{attribute 'GeneratedUsingTerminal: EK1100-0000-0018'}
{attribute addProperty BoxType "EK1100-0000-0018"}
{attribute addProperty Id "Beckhoff_APS1xxxEK1122Beckhoff_APS1xxxEK1122_47B4CB21266A_0002_APS1003_5000_0016APS1003_748FE0C1320"}
{attribute addProperty CRC "3524367647"}
{attribute addProperty Size "586"}
TYPE Beckhoff_APS1xxx_D211951F EXTENDS EK1100_AB5A9467 :
STRUCT
	{attribute addProperty Name "Beckhoff_APS1xxxEK1122"}
	{attribute addProperty PreviousPort "Beckhoff APS1xxx : B"}
	Beckhoff_APS1xxxEK1122 : Beckhoff_APS1xxxEK1122_47B4CB21;
	{attribute addProperty Name "A_0002_APS1003_5000_0016"}
	{attribute addProperty PreviousPort "Beckhoff APS1xxxEK1122 : C"}
	A_0002_APS1003_5000_0016 : APS1003_748FE0C1;
END_STRUCT
END_TYPE

(* stored: Version 1.2.0.0, ProductVersion 3.1.4024.9
   DUT Beckhoff_APS1xxx_D211951F: Id {4e013bb2-dd6b-494b-a621-0e9ea4602ede} *)
